    ENDPROC
    !The procedure below contains linear moves to draw the outline of letter G with predefined targets
    PROC LetterG()
        TPErase;
        MoveL Target_1310,v50,z5,PenTool\WObj:=A3paper;
        MoveL Target_1320,v50,fine,PenTool\WObj:=A3paper;
        MoveL Target_1330,v50,z5,PenTool\WObj:=A3paper;
        MoveC Target_1331,Target_1340,v50,z5,PenTool\WObj:=A3paper;
        MoveC Target_1341,Target_1350,v50,z5,PenTool\WObj:=A3paper;
        MoveC Target_1360,Target_1370,v50,z5,PenTool\WObj:=A3paper;
        MoveL Target_1380,v50,z5,PenTool\WObj:=A3paper;
        MoveL Target_1390,v50,z5,PenTool\WObj:=A3paper;
        MoveL Target_1400,v50,z5,PenTool\WObj:=A3paper;
        MoveC Target_1410,Target_1411,v50,z5,PenTool\WObj:=A3paper;
        MoveL Target_1420,v50,z10,PenTool\WObj:=A3paper;
        MoveC Target_1421,Target_1430,v50,z5,PenTool\WObj:=A3paper;
        MoveL Target_1480,v50,z5,PenTool\WObj:=A3paper;
        MoveL Target_1490,v50,z5,PenTool\WObj:=A3paper;
        MoveL Target_1500,v50,z5,PenTool\WObj:=A3paper;
        MoveL Target_1510,v50,z5,PenTool\WObj:=A3paper;
        MoveL Target_1520,v50,z5,PenTool\WObj:=A3paper;
        MoveL Target_1520,v50,z5,PenTool\WObj:=A3paper;
        MoveL Target_1530,v50,z5,PenTool\WObj:=A3paper;
        MoveL Target_1540,v50,z5,PenTool\WObj:=A3paper;
        MoveL Target_1560,v50,z5,PenTool\WObj:=A3paper;
        MoveL Target_1550,v50,z5,PenTool\WObj:=A3paper;
        MoveL Target_1570,v50,z5,PenTool\WObj:=A3paper;
        MoveL Target_1580,v50,z5,PenTool\WObj:=A3paper;
        MoveL Target_1600,v50,z5,PenTool\WObj:=A3paper;
        MoveL Target_1590,v50,z5,PenTool\WObj:=A3paper;
        MoveL Target_1600,v50,z100,PenTool\WObj:=A3paper;
        MoveL Target_1610,v50,z5,PenTool\WObj:=A3paper;
        MoveL Target_1620,v50,fine,PenTool\WObj:=A3paper;
        MoveL Target_1621,v50,z100,PenTool\WObj:=A3paper;
        home;
    ENDPROC
    !this procedure contains linear moves to draw the outline of letter M with predefined targets
    PROC letter_M()
        TPErase;
        MoveL Target_970,v50,z100,PenTool\WObj:=A3paper;
        MoveL Target_980,v50,z100,PenTool\WObj:=A3paper;
        MoveL Target_990,v50,z0,PenTool\WObj:=A3paper;
        MoveL Target_1000,v50,z100,PenTool\WObj:=A3paper;
        MoveL Target_1010,v50,z100,PenTool\WObj:=A3paper;
        MoveL Target_1020,v50,z100,PenTool\WObj:=A3paper;
        MoveL Target_1040,v50,z0,PenTool\WObj:=A3paper;
        MoveL Target_1050,v50,z0,PenTool\WObj:=A3paper;
        MoveL Target_1060,v50,z0,PenTool\WObj:=A3paper;
        MoveL Target_1070,v50,z0,PenTool\WObj:=A3paper;
        MoveL Target_1080,v50,z0,PenTool\WObj:=A3paper;
        MoveL Target_1090,v50,z0,PenTool\WObj:=A3paper;
        MoveL Target_1100,v50,z0,PenTool\WObj:=A3paper;
        MoveL Target_1120,v50,z100,PenTool\WObj:=A3paper;
        MoveL Target_1110,v50,z100,PenTool\WObj:=A3paper;
        MoveL Target_1130,v50,z100,PenTool\WObj:=A3paper;
        MoveL Target_1150,v50,z0,PenTool\WObj:=A3paper;
        MoveL Target_1140,v50,z100,PenTool\WObj:=A3paper;
        MoveL Target_1160,v50,z100,PenTool\WObj:=A3paper;
        MoveL Target_1180,v50,z0,PenTool\WObj:=A3paper;
        MoveL Target_1170,v50,z0,PenTool\WObj:=A3paper;
        MoveL Target_1200,v50,z100,PenTool\WObj:=A3paper;
        MoveL Target_1190,v50,z100,PenTool\WObj:=A3paper;
        MoveL Target_1210,v50,z0,PenTool\WObj:=A3paper;
        MoveL Target_1220,v50,z0,PenTool\WObj:=A3paper;
        MoveL Target_1230,v50,z0,PenTool\WObj:=A3paper;
        MoveL Target_1240,v50,z0,PenTool\WObj:=A3paper;
        MoveL Target_1250,v50,z100,PenTool\WObj:=A3paper;
        MoveL Target_1260,v50,z100,PenTool\WObj:=A3paper;
        MoveL Target_1270,v50,z0,PenTool\WObj:=A3paper;
        MoveL Target_1280,v50,z100,PenTool\WObj:=A3paper;
        MoveL Target_1290,v50,fine,PenTool\WObj:=A3paper;
        MoveL Target_1300,v50,z100,PenTool\WObj:=A3paper;
    ENDPROC
    !This procedure contains a joint move to move the robot to a position defined as home position
    PROC home()
        MoveJ Target_1630,v50,z100,PenTool\WObj:=A3paper;
    ENDPROC
    !This procedure contains linear moves to calibrate the position of an A3 paper(the workobject)
    PROC paperCalibration()
        MoveL Target_3760,v50,fine,PenTool\WObj:=A3paper;
        WaitTime 3;
        MoveL Target_3770,v50,fine,PenTool\WObj:=A3paper;
        WaitTime 3;
        MoveL Target_3780,v50,fine,PenTool\WObj:=A3paper;
        WaitTime 3;
        MoveL Target_3790,v50,fine,PenTool\WObj:=A3paper;
        WaitTime 3;
        MoveL Target_3800,v50,fine,PenTool\WObj:=A3paper;
        WaitTime 3;
    ENDPROC
    !This procedure contains linear moves to draw the outline of number one with predefined targets
    PROC number_1()
        MoveL Target_3810,v50,fine,PenTool\WObj:=A3paper;
        MoveL Target_3820,v50,fine,PenTool\WObj:=A3paper;
        MoveL Target_3830,v50,fine,PenTool\WObj:=A3paper;
        MoveL Target_3840,v50,fine,PenTool\WObj:=A3paper;
        MoveL Target_3850,v50,fine,PenTool\WObj:=A3paper;
        MoveL Target_3860,v50,fine,PenTool\WObj:=A3paper;
        MoveL Target_3870,v50,fine,PenTool\WObj:=A3paper;
        MoveL Target_3880,v50,fine,PenTool\WObj:=A3paper;
        MoveL Target_3890,v50,fine,PenTool\WObj:=A3paper;
        MoveL Target_3900,v50,fine,PenTool\WObj:=A3paper;
        MoveL Target_3910,v50,fine,PenTool\WObj:=A3paper;
    ENDPROC
    !This procedure contains linear moves to draw the outline of number two with predefined targets
    PROC number_2()
        MoveL Target_3920,v50,fine,PenTool\WObj:=A3paper;
        MoveL Target_3930,v50,fine,PenTool\WObj:=A3paper;
        MoveL Target_3940,v50,fine,PenTool\WObj:=A3paper;
        MoveL Target_3950,v50,fine,PenTool\WObj:=A3paper;
        MoveL Target_3960,v50,fine,PenTool\WObj:=A3paper;
        MoveL Target_3970,v50,fine,PenTool\WObj:=A3paper;
        MoveL Target_3980,v50,fine,PenTool\WObj:=A3paper;
        MoveL Target_3990,v50,fine,PenTool\WObj:=A3paper;
        MoveL Target_4000,v50,fine,PenTool\WObj:=A3paper;
        MoveL Target_4010,v50,fine,PenTool\WObj:=A3paper;
        MoveL Target_4020,v50,fine,PenTool\WObj:=A3paper;
        MoveL Target_4030,v50,fine,PenTool\WObj:=A3paper;
        MoveL Target_4040,v50,fine,PenTool\WObj:=A3paper;
        MoveL Target_4050,v50,fine,PenTool\WObj:=A3paper;
        MoveL Target_4060,v50,fine,PenTool\WObj:=A3paper;
        MoveL Target_4070,v50,fine,PenTool\WObj:=A3paper;
        MoveL Target_4080,v50,fine,PenTool\WObj:=A3paper;
        MoveL Target_4090,v50,fine,PenTool\WObj:=A3paper;
        MoveL Target_4100,v50,fine,PenTool\WObj:=A3paper;
        MoveL Target_4110,v50,fine,PenTool\WObj:=A3paper;
        MoveL Target_4120,v50,fine,PenTool\WObj:=A3paper;
        MoveL Target_4130,v50,fine,PenTool\WObj:=A3paper;
        MoveL Target_4140,v50,fine,PenTool\WObj:=A3paper;
        MoveL Target_4150,v50,fine,PenTool\WObj:=A3paper;
        MoveL Target_4160,v50,fine,PenTool\WObj:=A3paper;
    ENDPROC
    !This procedure contains linear moves to draw the outline of number three with predefined targets
    PROC number_3()
        MoveL Target_4170,v50,fine,PenTool\WObj:=A3paper;
        MoveL Target_4180,v50,fine,PenTool\WObj:=A3paper;
        MoveL Target_4190,v50,fine,PenTool\WObj:=A3paper;
        MoveL Target_4200,v50,fine,PenTool\WObj:=A3paper;
        MoveL Target_4210,v50,fine,PenTool\WObj:=A3paper;
        MoveL Target_4220,v50,fine,PenTool\WObj:=A3paper;
        MoveL Target_4230,v50,fine,PenTool\WObj:=A3paper;
        MoveL Target_4240,v50,fine,PenTool\WObj:=A3paper;
        MoveL Target_4250,v50,fine,PenTool\WObj:=A3paper;
        MoveL Target_4260,v50,fine,PenTool\WObj:=A3paper;
        MoveL Target_4270,v50,fine,PenTool\WObj:=A3paper;
        MoveL Target_4280,v50,fine,PenTool\WObj:=A3paper;
        MoveL Target_4290,v50,fine,PenTool\WObj:=A3paper;
        MoveL Target_4300,v50,fine,PenTool\WObj:=A3paper;
        MoveL Target_4310,v50,fine,PenTool\WObj:=A3paper;
        MoveL Target_4320,v50,fine,PenTool\WObj:=A3paper;
        MoveL Target_4330,v50,fine,PenTool\WObj:=A3paper;
        MoveL Target_4340,v50,fine,PenTool\WObj:=A3paper;
        MoveL Target_4350,v50,fine,PenTool\WObj:=A3paper;
        MoveL Target_4360,v50,fine,PenTool\WObj:=A3paper;
        MoveL Target_4370,v50,fine,PenTool\WObj:=A3paper;
        MoveL Target_4380,v50,fine,PenTool\WObj:=A3paper;
        MoveL Target_4390,v50,fine,PenTool\WObj:=A3paper;
        MoveL Target_4400,v50,fine,PenTool\WObj:=A3paper;
        MoveL Target_4410,v50,fine,PenTool\WObj:=A3paper;
    ENDPROC
    !This procedure contains linear moves to draw the outline of number four with predefined targets
    PROC number_4()
        MoveL Target_4420,v50,fine,PenTool\WObj:=A3paper;
        MoveL Target_4430,v50,fine,PenTool\WObj:=A3paper;
        MoveL Target_4440,v50,fine,PenTool\WObj:=A3paper;
        MoveL Target_4450,v50,fine,PenTool\WObj:=A3paper;
        MoveL Target_4460,v50,fine,PenTool\WObj:=A3paper;
        MoveL Target_4470,v50,fine,PenTool\WObj:=A3paper;
        MoveL Target_4480,v50,fine,PenTool\WObj:=A3paper;
        MoveL Target_4490,v50,fine,PenTool\WObj:=A3paper;
        MoveL Target_4500,v50,fine,PenTool\WObj:=A3paper;
        MoveL Target_4510,v50,fine,PenTool\WObj:=A3paper;
        MoveL Target_4520,v50,fine,PenTool\WObj:=A3paper;
        MoveL Target_4530,v50,fine,PenTool\WObj:=A3paper;
        MoveL Target_4540,v50,fine,PenTool\WObj:=A3paper;
        MoveL Target_4550,v50,fine,PenTool\WObj:=A3paper;
        MoveL Target_4560,v50,fine,PenTool\WObj:=A3paper;
        MoveL Target_4570,v50,fine,PenTool\WObj:=A3paper;
        MoveL Target_4571,v50,fine,PenTool\WObj:=A3paper;
        MoveL Target_4580,v50,fine,PenTool\WObj:=A3paper;
        MoveL Target_4590,v50,fine,PenTool\WObj:=A3paper;
        MoveL Target_4600,v50,fine,PenTool\WObj:=A3paper;
        MoveL Target_4610,v50,fine,PenTool\WObj:=A3paper;
    ENDPROC
    !This procedure contains linear moves to draw the outline of number five with predefined targets
    PROC number_5()
        MoveL Target_4620,v30,fine,PenTool\WObj:=A3paper;
        MoveL Target_4630,v30,fine,PenTool\WObj:=A3paper;
        MoveL Target_4640,v30,fine,PenTool\WObj:=A3paper;
        MoveL Target_4650,v30,fine,PenTool\WObj:=A3paper;
        MoveL Target_4660,v30,fine,PenTool\WObj:=A3paper;
        MoveL Target_4670,v30,fine,PenTool\WObj:=A3paper;
        MoveL Target_4680,v30,fine,PenTool\WObj:=A3paper;
        MoveL Target_4690,v30,fine,PenTool\WObj:=A3paper;
        MoveL Target_4700,v30,fine,PenTool\WObj:=A3paper;
        MoveL Target_4710,v30,fine,PenTool\WObj:=A3paper;
        MoveL Target_4720,v30,fine,PenTool\WObj:=A3paper;
        MoveL Target_4730,v30,fine,PenTool\WObj:=A3paper;
        MoveL Target_4740,v30,fine,PenTool\WObj:=A3paper;
        MoveL Target_4750,v30,fine,PenTool\WObj:=A3paper;
        MoveL Target_4760,v30,fine,PenTool\WObj:=A3paper;
        MoveL Target_4770,v30,fine,PenTool\WObj:=A3paper;
        MoveL Target_4780,v30,fine,PenTool\WObj:=A3paper;
        MoveL Target_4790,v30,fine,PenTool\WObj:=A3paper;
        MoveL Target_4800,v30,fine,PenTool\WObj:=A3paper;
        MoveL Target_4810,v30,fine,PenTool\WObj:=A3paper;
        MoveL Target_4820,v30,fine,PenTool\WObj:=A3paper;
        MoveL Target_4830,v30,fine,PenTool\WObj:=A3paper;
        MoveL Target_4840,v30,fine,PenTool\WObj:=A3paper;
        MoveL Target_4850,v30,fine,PenTool\WObj:=A3paper;
    ENDPROC
    !This procedure contains linear moves to draw the outline of number six with predefined targets
    PROC number_6()
        MoveL Target_4860,v50,fine,PenTool\WObj:=A3paper;
        MoveL Target_4870,v50,fine,PenTool\WObj:=A3paper;
        MoveL Target_4880,v50,fine,PenTool\WObj:=A3paper;
        MoveL Target_4890,v50,fine,PenTool\WObj:=A3paper;
        MoveL Target_4900,v50,fine,PenTool\WObj:=A3paper;
        MoveL Target_4910,v50,fine,PenTool\WObj:=A3paper;
        MoveL Target_4920,v50,fine,PenTool\WObj:=A3paper;
        MoveL Target_4930,v50,fine,PenTool\WObj:=A3paper;
        MoveL Target_4940,v50,fine,PenTool\WObj:=A3paper;
        MoveL Target_4950,v50,fine,PenTool\WObj:=A3paper;
        MoveL Target_4960,v50,fine,PenTool\WObj:=A3paper;
        MoveL Target_4970,v50,fine,PenTool\WObj:=A3paper;
        MoveL Target_4980,v50,fine,PenTool\WObj:=A3paper;
        MoveL Target_4990,v50,fine,PenTool\WObj:=A3paper;
        MoveL Target_5000,v50,fine,PenTool\WObj:=A3paper;
        MoveL Target_5010,v50,fine,PenTool\WObj:=A3paper;
        MoveL Target_5020,v50,fine,PenTool\WObj:=A3paper;
        MoveL Target_5030,v50,fine,PenTool\WObj:=A3paper;
        MoveL Target_5040,v50,fine,PenTool\WObj:=A3paper;
        MoveL Target_5050,v50,fine,PenTool\WObj:=A3paper;
        MoveL Target_5060,v50,fine,PenTool\WObj:=A3paper;
        MoveL Target_5070,v50,fine,PenTool\WObj:=A3paper;
        MoveL Target_5071,v50,fine,PenTool\WObj:=A3paper;
        MoveL Target_5080,v50,fine,PenTool\WObj:=A3paper;
        MoveL Target_5090,v50,fine,PenTool\WObj:=A3paper;
        MoveL Target_5100,v50,fine,PenTool\WObj:=A3paper;
        MoveL Target_5110,v50,fine,PenTool\WObj:=A3paper;
        MoveL Target_5120,v50,fine,PenTool\WObj:=A3paper;
        MoveL Target_5130,v50,fine,PenTool\WObj:=A3paper;
    ENDPROC
    !This procedure contains linear moves to draw the outline of number seven with predefined targets
    PROC number_7()
        MoveL Target_5140,v50,fine,PenTool\WObj:=A3paper;
        MoveL Target_5150,v50,fine,PenTool\WObj:=A3paper;
        MoveL Target_5160,v50,fine,PenTool\WObj:=A3paper;
        MoveL Target_5170,v50,fine,PenTool\WObj:=A3paper;
        MoveL Target_5180,v50,fine,PenTool\WObj:=A3paper;
        MoveL Target_5190,v50,fine,PenTool\WObj:=A3paper;
        MoveL Target_5200,v50,fine,PenTool\WObj:=A3paper;
        MoveL Target_5210,v50,fine,PenTool\WObj:=A3paper;
        MoveL Target_5220,v50,fine,PenTool\WObj:=A3paper;
        MoveL Target_5230,v50,fine,PenTool\WObj:=A3paper;
        MoveL Target_5240,v50,fine,PenTool\WObj:=A3paper;
        MoveL Target_5250,v50,fine,PenTool\WObj:=A3paper;
        MoveL Target_5260,v50,fine,PenTool\WObj:=A3paper;
        MoveL Target_5270,v50,fine,PenTool\WObj:=A3paper;
        MoveL Target_5280,v50,fine,PenTool\WObj:=A3paper;
        MoveL Target_5290,v50,fine,PenTool\WObj:=A3paper;
        MoveL Target_5300,v50,fine,PenTool\WObj:=A3paper;
        MoveL Target_5310,v50,fine,PenTool\WObj:=A3paper;
        MoveL Target_5320,v50,fine,PenTool\WObj:=A3paper;
        MoveL Target_5330,v50,fine,PenTool\WObj:=A3paper;
        MoveL Target_5340,v50,fine,PenTool\WObj:=A3paper;
    ENDPROC
    !This procedure contains linear moves to draw the outline of number eight with predefined targets
    PROC number_8()
        MoveL Target_5350,v50,fine,PenTool\WObj:=A3paper;
        MoveL Target_5360,v50,fine,PenTool\WObj:=A3paper;
        MoveL Target_5370,v50,fine,PenTool\WObj:=A3paper;
        MoveL Target_5380,v50,fine,PenTool\WObj:=A3paper;
        MoveL Target_5390,v50,fine,PenTool\WObj:=A3paper;
        MoveL Target_5400,v50,fine,PenTool\WObj:=A3paper;
        MoveL Target_5410,v50,fine,PenTool\WObj:=A3paper;
        MoveL Target_5420,v50,fine,PenTool\WObj:=A3paper;
        MoveL Target_5430,v50,fine,PenTool\WObj:=A3paper;
        MoveL Target_5440,v50,fine,PenTool\WObj:=A3paper;
        MoveL Target_5450,v50,fine,PenTool\WObj:=A3paper;
        MoveL Target_5460,v50,fine,PenTool\WObj:=A3paper;
        MoveL Target_5470,v50,fine,PenTool\WObj:=A3paper;
        MoveL Target_5480,v50,fine,PenTool\WObj:=A3paper;
        MoveL Target_5490,v50,fine,PenTool\WObj:=A3paper;
        MoveL Target_5500,v50,fine,PenTool\WObj:=A3paper;
        MoveL Target_5510,v50,fine,PenTool\WObj:=A3paper;
        MoveL Target_5520,v50,fine,PenTool\WObj:=A3paper;
        MoveL Target_5530,v50,fine,PenTool\WObj:=A3paper;
        MoveL Target_5540,v50,fine,PenTool\WObj:=A3paper;
        MoveL Target_5540_2,v50,fine,PenTool\WObj:=A3paper;
        MoveL Target_5610,v50,fine,PenTool\WObj:=A3paper;
        MoveL Target_5550,v50,fine,PenTool\WObj:=A3paper;
        MoveL Target_5560,v50,fine,PenTool\WObj:=A3paper;
        MoveL Target_5570,v50,fine,PenTool\WObj:=A3paper;
        MoveL Target_5580,v50,fine,PenTool\WObj:=A3paper;
        MoveL Target_5590,v50,fine,PenTool\WObj:=A3paper;
        MoveL Target_5600,v50,fine,PenTool\WObj:=A3paper;
        MoveL Target_5610,v50,fine,PenTool\WObj:=A3paper;
        MoveL Target_5610_2,v50,fine,PenTool\WObj:=A3paper;
        MoveL Target_5620,v50,fine,PenTool\WObj:=A3paper;
        MoveL Target_5630,v50,fine,PenTool\WObj:=A3paper;
        MoveL Target_5640,v50,fine,PenTool\WObj:=A3paper;
        MoveL Target_5650,v50,fine,PenTool\WObj:=A3paper;
        MoveL Target_5660,v50,fine,PenTool\WObj:=A3paper;
        MoveL Target_5670,v50,fine,PenTool\WObj:=A3paper;
        MoveL Target_5680,v50,fine,PenTool\WObj:=A3paper;
    ENDPROC
    !This procedure contains linear moves to draw the outline of number nine with predefined targets
    PROC number_9()
        MoveL Target_5690,v50,fine,PenTool\WObj:=A3paper;
        MoveL Target_5700,v50,fine,PenTool\WObj:=A3paper;
        MoveL Target_5710,v50,fine,PenTool\WObj:=A3paper;
        MoveL Target_5720,v50,fine,PenTool\WObj:=A3paper;
        MoveL Target_5730,v50,fine,PenTool\WObj:=A3paper;
        MoveL Target_5740,v50,fine,PenTool\WObj:=A3paper;
        MoveL Target_5750,v50,fine,PenTool\WObj:=A3paper;
        MoveL Target_5760,v50,fine,PenTool\WObj:=A3paper;
        MoveL Target_5770,v50,fine,PenTool\WObj:=A3paper;
        MoveL Target_5780,v50,fine,PenTool\WObj:=A3paper;
        MoveL Target_5790,v50,fine,PenTool\WObj:=A3paper;
        MoveL Target_5800,v50,fine,PenTool\WObj:=A3paper;
        MoveL Target_5810,v50,fine,PenTool\WObj:=A3paper;
        MoveL Target_5820,v50,fine,PenTool\WObj:=A3paper;
        MoveL Target_5830,v50,fine,PenTool\WObj:=A3paper;
        MoveL Target_5840,v50,fine,PenTool\WObj:=A3paper;
        MoveL Target_5860,v50,fine,PenTool\WObj:=A3paper;
        MoveL Target_5870,v50,fine,PenTool\WObj:=A3paper;
        MoveL Target_5880,v50,fine,PenTool\WObj:=A3paper;
        MoveL Target_5880_2,v50,fine,PenTool\WObj:=A3paper;
        MoveL Target_5890,v50,fine,PenTool\WObj:=A3paper;
        MoveL Target_5900,v50,fine,PenTool\WObj:=A3paper;
        MoveL Target_5910,v50,fine,PenTool\WObj:=A3paper;
        MoveL Target_5920,v50,fine,PenTool\WObj:=A3paper;
        MoveL Target_5930,v50,fine,PenTool\WObj:=A3paper;
        MoveL Target_5940,v50,fine,PenTool\WObj:=A3paper;
        MoveL Target_5950,v50,fine,PenTool\WObj:=A3paper;
        MoveL Target_5960,v50,fine,PenTool\WObj:=A3paper;
        MoveL Target_5850,v50,fine,PenTool\WObj:=A3paper;
    ENDPROC
    !This procedure contains linear moves to draw the outline of number zero with predefined targets
    PROC number_0()
        MoveL Target_5970,v50,fine,PenTool\WObj:=A3paper;
        MoveL Target_5980,v50,fine,PenTool\WObj:=A3paper;
        MoveL Target_5990,v50,fine,PenTool\WObj:=A3paper;
        MoveL Target_6000,v50,fine,PenTool\WObj:=A3paper;
        MoveL Target_6010,v50,fine,PenTool\WObj:=A3paper;
        MoveL Target_6020,v50,fine,PenTool\WObj:=A3paper;
        MoveL Target_6030,v50,fine,PenTool\WObj:=A3paper;
        MoveL Target_6040,v50,fine,PenTool\WObj:=A3paper;
        MoveL Target_6050,v50,fine,PenTool\WObj:=A3paper;
        MoveL Target_6060,v50,fine,PenTool\WObj:=A3paper;
        MoveL Target_6070,v50,fine,PenTool\WObj:=A3paper;
        MoveL Target_6080,v50,fine,PenTool\WObj:=A3paper;
        MoveL Target_6090,v50,fine,PenTool\WObj:=A3paper;
        MoveL Target_6100,v50,fine,PenTool\WObj:=A3paper;
        MoveL Target_6110,v50,fine,PenTool\WObj:=A3paper;
        MoveL Target_6110_2,v50,fine,PenTool\WObj:=A3paper;
        MoveL Target_6120,v50,fine,PenTool\WObj:=A3paper;
        MoveL Target_6130,v50,fine,PenTool\WObj:=A3paper;
        MoveL Target_6140,v50,fine,PenTool\WObj:=A3paper;
        MoveL Target_6150,v50,fine,PenTool\WObj:=A3paper;
        MoveL Target_6160,v50,fine,PenTool\WObj:=A3paper;
        MoveL Target_6170,v50,fine,PenTool\WObj:=A3paper;
        MoveL Target_6180,v50,fine,PenTool\WObj:=A3paper;
        MoveL Target_6190,v50,fine,PenTool\WObj:=A3paper;
        MoveL Target_6200,v50,z100,PenTool\WObj:=A3paper;
    ENDPROC
    !This procedure contains the path of to draw letter M and G( My initials)
    PROC DRAW_INITIALS()
        letter_M;
        LetterG;

    ENDPROC
    PROC manualJoggin()
        MoveL Target_6290,v50,fine,PenTool\WObj:=A3paper;
        MoveL Target_6300,v50,fine,PenTool\WObj:=A3paper;
        MoveL Target_6310,v50,fine,PenTool\WObj:=A3paper;
        MoveL Target_6320,v50,fine,PenTool\WObj:=A3paper;
        MoveL Target_6330,v50,fine,PenTool\WObj:=A3paper;
    ENDPROC
ENDMODULE
